INTERFACE I_XtsProcess_Station

END_INTERFACE

(* stored: Version 1.1.0.1, ProductVersion 3.1.4024.15
   Itf I_XtsProcess_Station: Id {7e6974e1-9081-4369-af45-d77e111a3519} *)
